SUBAPPLICATION ACTION_CLIENT_FEEDBACK_MESSAGE (* Subapplication Type *)
  (* Standard: 61499-2 *)
  (* Version 1.0, 2023-03-23, derPi *)
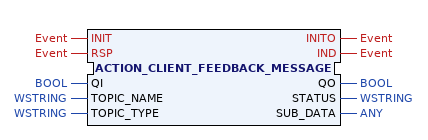
  EVENT_INPUT
    INIT; (* Initialization Request *)
    RSP;
  END_EVENT
  EVENT_OUTPUT
    INITO; (* Initialization Confirm *)
    IND;
  END_EVENT
  VAR_INPUT
    QI : BOOL; (* Input event qualifier *)
    TOPIC_NAME : WSTRING;
    TOPIC_TYPE : WSTRING;
  END_VAR
  VAR_OUTPUT
    QO : BOOL; (* Output event qualifier *)
    STATUS : WSTRING;
    SUB_DATA : ANY;
  END_VAR
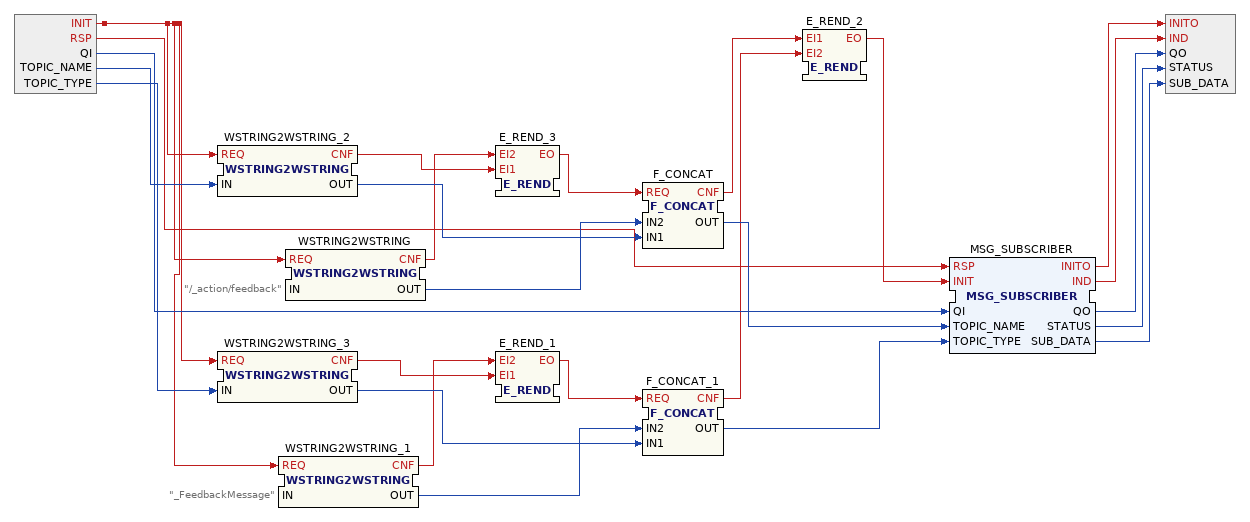
  FBS
    WSTRING2WSTRING_3 : WSTRING2WSTRING;
    F_CONCAT_1 : F_CONCAT;
    E_REND_1 : E_REND;
    WSTRING2WSTRING_1 : WSTRING2WSTRING(IN := "_FeedbackMessage");
    WSTRING2WSTRING_2 : WSTRING2WSTRING;
    E_REND_2 : E_REND;
    WSTRING2WSTRING : WSTRING2WSTRING(IN := "/_action/feedback");
    E_REND_3 : E_REND;
    F_CONCAT : F_CONCAT;
  END_FBS
  SUBAPPS
    MSG_SUBSCRIBER : MSG_SUBSCRIBER;
  END_SUBAPPS
  EVENT_CONNECTIONS
    F_CONCAT.CNF TO E_REND_2.EI1;
    F_CONCAT_1.CNF TO E_REND_2.EI2;
    WSTRING2WSTRING_1.CNF TO E_REND_1.EI2;
    WSTRING2WSTRING.CNF TO E_REND_3.EI2;
    WSTRING2WSTRING_3.CNF TO E_REND_1.EI1;
    E_REND_1.EO TO F_CONCAT_1.REQ;
    E_REND_3.EO TO F_CONCAT.REQ;
    WSTRING2WSTRING_2.CNF TO E_REND_3.EI1;
    INIT TO WSTRING2WSTRING_2.REQ;
    INIT TO WSTRING2WSTRING.REQ;
    INIT TO WSTRING2WSTRING_3.REQ;
    INIT TO WSTRING2WSTRING_1.REQ;
    RSP TO MSG_SUBSCRIBER.RSP;
    E_REND_2.EO TO MSG_SUBSCRIBER.INIT;
    MSG_SUBSCRIBER.INITO TO INITO;
    MSG_SUBSCRIBER.IND TO IND;
  END_CONNECTIONS
  DATA_CONNECTIONS
    WSTRING2WSTRING.OUT TO F_CONCAT.IN2;
    WSTRING2WSTRING_2.OUT TO F_CONCAT.IN1;
    WSTRING2WSTRING_1.OUT TO F_CONCAT_1.IN2;
    WSTRING2WSTRING_3.OUT TO F_CONCAT_1.IN1;
    TOPIC_NAME TO WSTRING2WSTRING_2.IN;
    TOPIC_TYPE TO WSTRING2WSTRING_3.IN;
    QI TO MSG_SUBSCRIBER.QI;
    F_CONCAT.OUT TO MSG_SUBSCRIBER.TOPIC_NAME;
    F_CONCAT_1.OUT TO MSG_SUBSCRIBER.TOPIC_TYPE;
    MSG_SUBSCRIBER.QO TO QO;
    MSG_SUBSCRIBER.STATUS TO STATUS;
    MSG_SUBSCRIBER.SUB_DATA TO SUB_DATA;
  END_CONNECTIONS
END_SUBAPPLICATION
